{attribute 'linkalways'} 
{attribute 'no_explicit_call' := 'This FB is a CLASS and must be accessed using methods or properties'}
{attribute 'enable_dynamic_creation'}
FUNCTION_BLOCK _ETcVnPixelEncoding EXTENDS EnumDatatypeBase
VAR
	localData : ETcVnPixelEncoding;
	activeData : REFERENCE TO ETcVnPixelEncoding;
	enumBaseDatatype : _BYTE(localData);
END_VAR

METHOD PRIVATE AddLocalEnumeration
VAR_INPUT
	Enumeration : T_MAXSTRING;
	Value : ETcVnPixelEncoding;
END_VAR
AddEnumeration(Enumeration, Value);
END_METHOD

PROPERTY PUBLIC Address : PVOID
GET
Address := ADR(activeData);
END_GET
END_PROPERTY

METHOD PUBLIC ClearReference
VAR_INPUT
END_VAR
activeData REF= localData;
SetBaseDatatypeReference();
END_METHOD

METHOD PUBLIC Clone : I_Datatype
VAR
    pClone : POINTER TO _ETcVnPixelEncoding;
END_VAR
pClone := __NEW(_ETcVnPixelEncoding(InitialValue := Value));
Clone := pClone^;
END_METHOD

METHOD FB_init : BOOL
VAR_INPUT
	bInitRetains : BOOL; // if TRUE, the retain variables are initialized (warm start / cold start)
	bInCopyCode : BOOL;  // if TRUE, the instance afterwards gets moved into the copy code (online change)
	InitialValue : ETcVnPixelEncoding;
END_VAR
localData := InitialValue;
AddBaseDatatype(enumBaseDatatype);
ClearReference();

AddLocalEnumeration('TCVN_PE_NONE', ETcVnPixelEncoding.TCVN_PE_NONE);
AddLocalEnumeration('TCVN_PE_BAYER_GR', ETcVnPixelEncoding.TCVN_PE_BAYER_GR);
AddLocalEnumeration('TCVN_PE_BAYER_RG', ETcVnPixelEncoding.TCVN_PE_BAYER_RG);
AddLocalEnumeration('TCVN_PE_BAYER_GB', ETcVnPixelEncoding.TCVN_PE_BAYER_GB);
AddLocalEnumeration('TCVN_PE_BAYER_BG', ETcVnPixelEncoding.TCVN_PE_BAYER_BG);
AddLocalEnumeration('TCVN_PE_YUV_411_UYYVYY', ETcVnPixelEncoding.TCVN_PE_YUV_411_UYYVYY);
AddLocalEnumeration('TCVN_PE_YUV_422_UYVY', ETcVnPixelEncoding.TCVN_PE_YUV_422_UYVY);
AddLocalEnumeration('TCVN_PE_YUV_422_YUYV', ETcVnPixelEncoding.TCVN_PE_YUV_422_YUYV);
AddLocalEnumeration('TCVN_PE_YCBCR_411_CBYYCRYY', ETcVnPixelEncoding.TCVN_PE_YCBCR_411_CBYYCRYY);
AddLocalEnumeration('TCVN_PE_YCBCR_422_CBYCRY', ETcVnPixelEncoding.TCVN_PE_YCBCR_422_CBYCRY);
AddLocalEnumeration('TCVN_PE_YCBCR_422_YCBYCR', ETcVnPixelEncoding.TCVN_PE_YCBCR_422_YCBYCR);
END_METHOD

PROPERTY PUBLIC Identifier : T_MAXSTRING
GET
Identifier := 'ETcVnPixelEncoding';
END_GET
END_PROPERTY

METHOD IsEnumeratorValueEqual : BOOL
VAR_INPUT
	Enumerator : I_KeyValueForwardEnumerator;
END_VAR
VAR
	storedValue : ETcVnPixelEncoding;
END_VAR
IF NOT Enumerator.TryGet(storedValue) THEN
	RETURN;
END_IF

IsEnumeratorValueEqual := storedValue = activeData;
END_METHOD

METHOD PUBLIC MakeReferenceTo
VAR_INPUT
	ReferenceTarget : REFERENCE TO ETcVnPixelEncoding;
END_VAR
activeData REF= ReferenceTarget;
SetBaseDatatypeReference();
END_METHOD

METHOD PROTECTED SetBaseDatatypeReference
VAR_INPUT
END_VAR
enumBaseDatatype.MakeReferenceTo(activeData);
END_METHOD

PROPERTY PUBLIC Size : UDINT
GET
Size := SIZEOF(activeData);
END_GET
END_PROPERTY

METHOD TryMakeReferenceTo : BOOL
VAR_INPUT
	Target : I_Datatype;
END_VAR
VAR
	targetAsEnum : I_EnumDatatype;
	pTargetData : POINTER TO ETcVnPixelEncoding;
END_VAR
IF NOT Target.TryResolveAsEnumDatatype(targetAsEnum) THEN
	RETURN;
END_IF

IF targetAsEnum.Identifier <> Identifier THEN
	RETURN;
END_IF

pTargetData := Target.Address;
activeData REF= pTargetData^;
SetBaseDatatypeReference();
TryMakeReferenceTo := TRUE;
END_METHOD

PROPERTY PUBLIC Value : ETcVnPixelEncoding
GET
Value := activeData;
END_GET
SET
activeData := Value;
END_SET
END_PROPERTY

END_FUNCTION_BLOCK

(* stored: Version 1.1.0.1, ProductVersion 3.1.4024.12
   POU _ETcVnPixelEncoding: Id {6c8cd06f-3019-44c4-93c7-3ae1434aef9f}, SpecialFunc None
   Folder Constructor: Id {c8e8eddf-89fb-4583-9083-c17631bf99dc}
   Folder Private: Id {e8210ae7-9a7b-4dc4-b76d-ffe5c1e2276f}
   Folder Protected: Id {d0349e2b-dc79-4906-bfd2-e5c863064813}
   Method AddLocalEnumeration: Id {f33ec11f-ec91-44e7-9a3a-bd8f31c6a4ca}
   Property Address: Id {02bb4169-1ee0-4ce3-b331-3bc8f5b688fe}
   Get Get: Id {03784653-d415-487c-912a-7f9ec249465b}
   Method ClearReference: Id {00a985dc-a86d-4460-bc67-9508d68e7cd4}
   Method Clone: Id {a910d5a1-8c7c-4aae-b123-2f5cd4d9c0b0}
   Method FB_init: Id {eac57cef-b529-423d-9df8-ea5dd4a392a5}
   Property Identifier: Id {c68bc1b9-7569-4288-8438-d36bbbd0084c}
   Get Get: Id {2b780a1c-6780-4ba2-a717-1faf4fb6212b}
   Method IsEnumeratorValueEqual: Id {36ff3683-1967-4f73-afb0-1d6cce9104bd}
   Method MakeReferenceTo: Id {e5af0996-d46d-410c-a803-ea3b50d7d055}
   Method SetBaseDatatypeReference: Id {5dbf0ef7-805c-4296-85ab-f3020aea2118}
   Property Size: Id {128e7c3b-60b2-4545-9b2d-82b89d89cc75}
   Get Get: Id {365cb414-1338-42f5-83cf-f49096e06194}
   Method TryMakeReferenceTo: Id {b169ec70-5f01-4344-ad6c-b80d4cf861e9}
   Property Value: Id {d44ae1cd-44de-4169-bd42-f82336da2541}
   Get Get: Id {498beab1-5133-4351-aed2-98b0bff89702}
   Set Set: Id {9aed7ede-95a8-4338-8497-0a323fd2cb7f} *)
